INTERFACE I_File

METHOD PUBLIC M_Append : BOOL
VAR_INPUT
	sText:			STRING(255);
END_VAR
END_METHOD

METHOD PUBLIC M_Close : BOOL
VAR_INPUT
END_VAR
END_METHOD

METHOD PUBLIC M_Create : BOOL
VAR_INPUT
	sPathName:		T_MaxString;
END_VAR
END_METHOD

METHOD PUBLIC M_Delete : BOOL
VAR_INPUT
	sPathName:		T_MaxString;
END_VAR
END_METHOD

METHOD PUBLIC M_Load : BOOL
VAR_INPUT
	sPathName:		T_MaxString;
	pData:			PVOID;
	nData:			UDINT;
END_VAR
END_METHOD

METHOD PUBLIC M_Open : BOOL
VAR_INPUT
	sPathName:		T_MaxString;
END_VAR
END_METHOD

METHOD PUBLIC M_Read : BOOL
VAR_INPUT
	pData:		PVOID;
	nData:		udint;
END_VAR
END_METHOD

METHOD PUBLIC M_Write : BOOL
VAR_INPUT
	pData:		POINTER TO BYTE;
	nData:		UDINT;
END_VAR
END_METHOD

PROPERTY PUBLIC P_Error : E_AdsError
GET
END_GET
END_PROPERTY

END_INTERFACE

(* stored: Version 1.1.0.1
   Itf I_File: Id {a333c476-be74-00f0-3a80-a82b3c3d9aac}
   Method M_Append: Id {fbb15c1d-2df5-0e39-2358-fb7bc74a9fc3}
   Method M_Close: Id {9ca2b871-cea1-0cae-0c40-7f2f8ac18932}
   Method M_Create: Id {62be88b4-a419-01a4-3b43-ca7984336fe9}
   Method M_Delete: Id {e4656072-e375-0752-19f3-361e4f242d1d}
   Method M_Load: Id {ea60e964-c358-0745-2adc-afecd745c703}
   Method M_Open: Id {050d30ac-1147-020e-09c2-cea6558cdf69}
   Method M_Read: Id {d6544e38-9389-075a-15aa-5bab85948640}
   Method M_Write: Id {ade87bcf-1dc4-0b90-0279-e8b498b630a0}
   Property P_Error: Id {bc44daab-bd44-0bcc-12e7-c5e0e48215a2}
   Get Get: Id {a52d3697-97be-4baa-bcef-0b8888c9b6b3} *)
